(* poll TCP Server for incoming data, transfer to standard string *)
FUNCTION_BLOCK FB_TCP_ReceiveString
VAR_INPUT
	bEnable				: BOOL;			(* set TRUE to enable periodic TCP data receive *)
	hSocket				: T_HSocket;	(* TCP socket *)
	tUpdateTime			: TIME;			(* receive update rate *)
	nSyncOffset			: DINT;			(* ms offset to spread TCP Server access loading *)
END_VAR
VAR_IN_OUT
	strTCPRxString		: T_MaxString;	(* string to which incoming TCP data will be appended *)
END_VAR
VAR_OUTPUT
	bDone				: BOOL;			(* TRUE = complete *)
	bBusy				: BOOL;			(* TRUE = in progress *)
	bError 				: BOOL;			(* TRUE = error *)
	nErrorID			: UDINT;		(* error code *)
	bDataReceived		: BOOL;			(* TRUE = data received *)
END_VAR
VAR
	fbTimer				: FB_PulseGenerator_Sync;
	bTCPReceive			: BOOL;
	nMaxBytes			: UDINT;
	fbTCPReceive		: FB_SocketReceive;
	strTCPRxChars		: T_MaxString;
END_VAR
(*
-------------------------------------------------------------------------------------------------
Date		Version	Author	Comments
-------------------------------------------------------------------------------------------------
30/01/2015	3.00.00	PB		Data received from TCP port every tUpdateTime secs
							nSyncTime allows access to TCP Server to be staggered and spread PLC task times

-------------------------------------------------------------------------------------------------
06/05/2013	1.43.01	PB		Chars received from TCP Server are now limited to the space available in strTCPData
16/08/2012	1.40.02	PB		Initial release
-------------------------------------------------------------------------------------------------
*)

(* TCP update timer *)
fbTimer(
	bEnable		:= bEnable,
	tPeriod		:= tUpdateTime,
	nSyncOffset	:= nSyncOffset
);

(* TCP update timer elapsed and fbTCPReceive is not active *)
IF fbTimer.bOutput = TRUE THEN

	(* max number of bytes that can be received into strTCPRxString on next cycle *)
	nMaxBytes := SIZEOF(strTCPRxString) - LEN2(ADR(strTCPRxString)) - 1;

	(* clear strTCPRxChars *)
	MEMSET(ADR(strTCPRxChars), 16#00, SIZEOF(strTCPRxChars));

	(* strTCPRxString has space for 1 or more bytes *)
	IF nMaxBytes > 0 THEN

		(* receive data from TCP port *)
		bTCPReceive := TRUE;
		bBusy := TRUE;
	END_IF

	(* clear outputs *)
	bDone := FALSE;
	bError := FALSE;
	nErrorID := 0;
	bDataReceived := FALSE;

(* TPC receive not active *)
ELSIF bTCPReceive = FALSE THEN

	(* clear outputs *)
	bDone := FALSE;
	bBusy := FALSE;
	bError := FALSE;
	nErrorID := 0;
	bDataReceived := FALSE;
END_IF


(* receive data from TCP server, max length determined by free chars available in strTCPData *)
fbTCPReceive(
	sSrvNetId	:= '',
	hSocket		:= hSocket,
	cbLen		:= nMaxBytes,
	pDest		:= ADR(strTCPRxChars),
	bExecute	:= bTCPReceive,
	tTimeout	:= T#500ms,
	bBusy		=> bBusy
);


(* receive TCP data complete *)
IF bTCPReceive = TRUE AND fbTCPReceive.bBusy = FALSE THEN

	(* receive TCP data completed OK *)
	IF fbTCPReceive.bError = FALSE THEN

		(* data bytes received *)
		IF fbTCPReceive.nRecBytes > 0 THEN

			(* append returned data to TCP data string *)
			strTCPRxString := CONCAT(strTCPRxString, strTCPRxChars);
			bDataReceived := TRUE;
		END_IF

	(* receive data error *)
	ELSE

		bDataReceived := FALSE;
		bError := TRUE;
		nErrorID := fbTCPReceive.nErrId;
	END_IF

	(* reset TCP receive flag *)
	bTCPReceive := FALSE;

	bDone := TRUE;
	bBusy := FALSE;

	(* close off fbReceiveTCPData *)
	fbTCPReceive(bExecute := FALSE);
END_IF

END_FUNCTION_BLOCK

(* stored: Version 1.1.0.1
   POU FB_TCP_ReceiveString: Id {205a0a87-5d47-4936-8366-0d0f3ec69e45}, SpecialFunc None *)
